// TIA Portal V20 export
// export: Created 2026-04-11T06:02:30.3925699Z, ExportSetting WithDefaults, DisplayName Totally Integrated Automation Portal, DisplayVersion V20, DisplayName TIA Portal Openness, DisplayVersion V20, DisplayName TIA Portal Version Control Interface, DisplayVersion V20, DisplayName STEP 7 Professional, DisplayVersion V20, DisplayName STEP 7 Safety, DisplayVersion V20, DisplayName WinCC Basic/Comfort/Advanced, DisplayVersion V20, DisplayName WinCC Unified, DisplayVersion V20
TYPE "udtHMI_MicroMotion"
// stored: IsFailsafeCompliant false
   STRUCT
      rTotal { ExternalWritable := 'False'} : Real;   // Total
      rFlow { ExternalWritable := 'False'} : Real;   // Actual flow
      rTemperature { ExternalWritable := 'False'} : Real;   // Actual Temperature
      rDensity { ExternalWritable := 'False'} : Real;   // Actual Density
      iErrorCode { ExternalWritable := 'False'} : Int;   // Error Code
      bPBEN_ResetTotal { ExternalWritable := 'False'} : Bool;   // Enable reset total button
      bPBEN_ResetError { ExternalWritable := 'False'} : Bool;   // Reset button enable
      bPB_ResetTotal : Bool;   // Reset total button
      bPB_ResetError : Bool;   // Reset error button
      bError { ExternalWritable := 'False'} : Bool;   // Error active
   END_STRUCT;
END_TYPE
